(* CODESYS project Übung4.project

Project tree, tasks and I/O mapping:
  CODESYS_Control_Win_V3 : CODESYS Control Win V3, 3S - Smart Software Solutions GmbH, version 3.5.3.60
    application Application
      libraries: Standard, 3.5.2.0 (System)
      task VISU_TASK (cyclic, interval 100 ms, priority 30) calls VisuElems.Visu_Prg
      task MainTask (cyclic, interval t#20ms, priority 1) calls Ampel
      program Ampel [LD]
      visualisation Ampel_Vis
  text list GlobalTextList
*)

// CODESYS_Control_Win_V3/Application/Ampel
PROGRAM Ampel
VAR
	rechts: BOOL;
	links: BOOL;
	Auto_Gelb: BOOL;
	Auto_Gruen: BOOL := TRUE;
	Ampel_Merker: BOOL;
	GelbPhase: TON;
	Auto_Rot: BOOL;
	Fussg_Gruen: BOOL;
	Fussg_Rot: BOOL := TRUE;
	GruenPhase: TON;
	RotPhase: TON;
	GelbPhase2: TON;
	Wait: TON;
END_VAR
VAR // added by the converter: edge detectors and wires of the graphical bodies
    _w1, _w2 : BOOL;
END_VAR

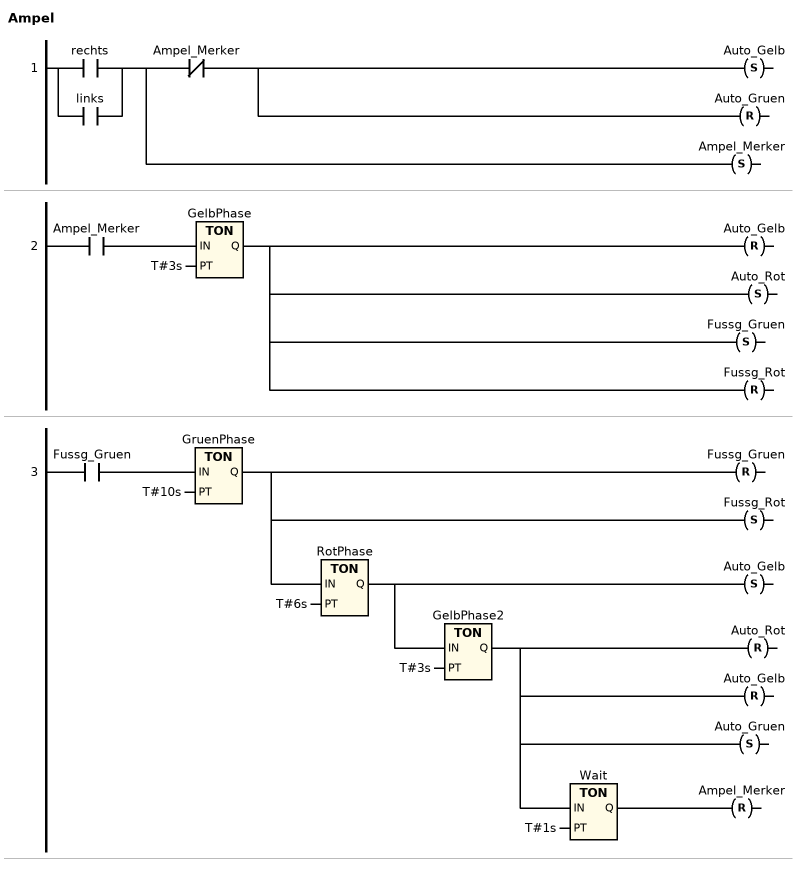
// NETWORK 1
_w1 := rechts OR links;
_w2 := _w1 AND NOT Ampel_Merker;
Auto_Gelb S= _w2;
Auto_Gruen R= _w2;
Ampel_Merker S= _w1;

// NETWORK 2
GelbPhase(IN := Ampel_Merker, PT := T#3s); // TON
Auto_Gelb R= GelbPhase.Q;
Auto_Rot S= GelbPhase.Q;
Fussg_Gruen S= GelbPhase.Q;
Fussg_Rot R= GelbPhase.Q;

// NETWORK 3
GruenPhase(IN := Fussg_Gruen, PT := T#10s); // TON
Fussg_Gruen R= GruenPhase.Q;
Fussg_Rot S= GruenPhase.Q;
RotPhase(IN := GruenPhase.Q, PT := T#6s); // TON
Auto_Gelb S= RotPhase.Q;
GelbPhase2(IN := RotPhase.Q, PT := T#3s); // TON
Auto_Rot R= GelbPhase2.Q;
Auto_Gelb R= GelbPhase2.Q;
Auto_Gruen S= GelbPhase2.Q;
Wait(IN := GelbPhase2.Q, PT := T#1s); // TON
Ampel_Merker R= Wait.Q;

END_PROGRAM

// CODESYS_Control_Win_V3/Application/Ampel_Vis
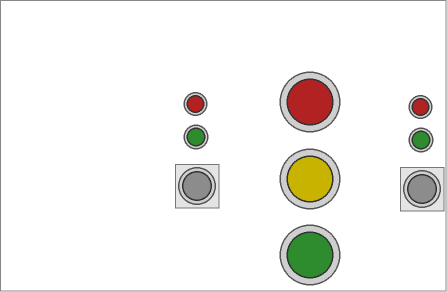
VISUALIZATION Ampel_Vis  // 447x292
    Lamp1 (182,90 27x28), variable: Ampel.Fussg_Rot, style: Lamp-Lamp1-Red
    Lamp1 (181,123 30x28), variable: Ampel.Fussg_Gruen, style: Lamp-Lamp1-Green
    Lamp1 (275,67 70x70), variable: Ampel.Auto_Rot, style: Lamp-Lamp1-Red
    Lamp1 (275,144 70x70), variable: Ampel.Auto_Gelb, style: Lamp-Lamp1-Yellow
    Lamp1 (275,220 70x70), variable: Ampel.Auto_Gruen, style: Lamp-Lamp1-Green
    PushSwitch (174,164 46x44), variable: Ampel.links, behaviour: TOGGLE, style: Switch-PushSwitch-Gray
    Lamp1 (407,93 27x28), variable: Ampel.Fussg_Rot, style: Lamp-Lamp1-Red
    Lamp1 (406,126 30x28), variable: Ampel.Fussg_Gruen, style: Lamp-Lamp1-Green
    PushSwitch (399,167 46x44), variable: Ampel.rechts, behaviour: TOGGLE, style: Switch-PushSwitch-Gray
END_VISUALIZATION
